TYPE Error_Handler_typ :
	STRUCT
		//ErrorHandler 	: ERR_HANDLER_typ;
		//ErrorInfo 	: ERR_TASK_INFO_typ;
	END_STRUCT
END_TYPE

(* stored: Version 1.1.0.1, ProductVersion 3.1.4024.3
   DUT Error_Handler_typ: Id {be2e9d25-416c-0aad-089a-69124a322209} *)
